{attribute 'GeneratedUsingTerminal: EL9222-4433-0018'}
{attribute addProperty BoxType "EL9222-4433-0018"}
{attribute addProperty Id "StatusAT %I*Status_FCAFFB9E11"}
{attribute addProperty CRC "2362336763"}
{attribute addProperty Size "11"}
TYPE OCP_Inputs_Channel_8CCE65FB EXTENDS InputBase_8311D824 :
STRUCT
	{attribute addProperty Name "Status"}
	Status AT %I* : Status_FCAFFB9E;
END_STRUCT
END_TYPE

(* stored: Version 1.2.0.0, ProductVersion 3.1.4024.9
   DUT OCP_Inputs_Channel_8CCE65FB: Id {920928f0-c6ac-452f-b305-1fd593e7b4b0} *)
